PROGRAM INTERNAL PRG_TEST
VAR
    _buttonPress_Test        : ButtonPress_Test;
    _buttonTrig_Test         : ButtonTrig_Test;
    _cylinderMonostable_Test : CylinderMonostable_Test;
    _cylinderBistable_Test   : CylinderBistable_Test;
END_VAR

TcUnit.RUN();

END_PROGRAM

(* stored: Version 1.1.0.1, ProductVersion 3.1.4024.12
   POU PRG_TEST: Id {f7b1802e-84ab-4d4a-a7d7-75643092ae7d}, SpecialFunc None *)
